FUNCTION_BLOCK FieldConnector (* Composite Function Block Type *)
  (* Standard: 61499-2 *)
  (* Version 0.0, 5/26/2025, Guillaume De Martino, Schneider Electric, template *)
  PACKAGE Main;
  (* 0 - INITIALIZATION *)
  (* 1 - FUNCTIONAL PARENT INTERFACE *)
  (* 3.A - TO THE FIELD INTERFACE *)
  (* 3.B - FROM THE FIELD INTERFACE *)
  (* AI *)
  (* DI *)
  (* AO *)
  (* DO *)
  (* OTHER DIRECT INPUT *)
  (* OTHER DIRECT OUTPUT *)
END_FUNCTION_BLOCK
